INTERFACE I_HasError

{attribute 'monitoring':='call'}
// Returns TRUE if an error has occurred
PROPERTY Error : BOOL
GET
END_GET
END_PROPERTY

END_INTERFACE

(* stored: Version 1.1.0.1, ProductVersion 3.1.4024.14
   Itf I_HasError: Id {38fbeb26-2e17-01ba-1b07-91aadc9f4503}
   Property Error: Id {2153587d-7715-0761-2820-f511a3974beb}
   Get Get: Id {db763451-fa61-009a-2ce3-90f31fd10e97} *)
